{attribute 'qualified_only'}
VAR_GLOBAL
	valve01: DUT_VALVE;
	ioValve01: DUT_IO;
	valve02: DUT_VALVE;
	ioValve02: DUT_IO;
END_VAR

VAR_GLOBAL CONSTANT
	STS_UNDEFINED : INT := 0;
	STS_CLOSED : INT := 10;
	STS_OPENING : INT := 20;
	STS_OPEN : INT := 30;
	STS_CLOSING : INT := 40;
END_VAR

(* stored: Version 1.1.0.1, ProductVersion 3.1.4024.12
   GVL GVL_VCM: Id {7721cf77-02c3-47c4-8ee5-866c25ff17d2} *)
